FUNCTION F_ReplaceLongSingleChar : T_LongSTRING
VAR_INPUT
	sFullCode		: T_LongSTRING;
	sCharRemove			: T_Char := '$1D';
	sReplacmentChar		: T_Char := '';
END_VAR
VAR
	sCodeSize		: STRING;
END_VAR

WHILE FIND2(ADR(sFullCode), ADR(sCharRemove)) > 0 DO
	REPLACE2(ADR(sFullCode),ADR(sReplacmentChar), ADR(sFullCode), 
						SIZEOF(sFullCode), LEN2(ADR(sCharRemove)), FIND2(ADR(sFullCode), ADR(sCharRemove)));
END_WHILE

(*Diagnostic part for long stirng operation *)
//sCodeSize := TO_STRING(LEN2(ADR(sFullCode)));
//CONCAT2(ADR(sCodeSize), ADR('_'), ADR(sCodeSize), SIZEOF(sCodeSize));	
//INSERT2(ADR(sFullCode), ADR(sCodeSize), ADR(sFullCode), SIZEOF(sFullCode), 0);
	
F_ReplaceLongSingleChar	:= sFullCode;

END_FUNCTION

(* stored: Version 1.1.0.1
   POU F_ReplaceLongSingleChar: Id {be285700-9975-40ba-924a-f5ee18996829}, SpecialFunc None *)
